(* IEC 61131-3 sources: programs/VI-54/VI-54_20171205/VI-54_20171205/Stations/Screen/LseClass170718/Class/DiagnosticStation, 1 file *)

(* ---- DiagnosticStation.st ---- *)
(*!
<Class
	Name               = "DiagnosticStation"
	Revision           = "1.1"
	RealtimeTask       = "false"
	CyclicTask         = "false"
	BackgroundTask     = "false"
	Sigmatek           = "false"
	OSInterface        = "false"
	HighPriority       = "false"
	Automatic          = "false"
	UpdateMode         = "Prescan"
	SharedCommandTable = "true"
	Objectsize         = "(960,420)"
	Comment            = "Use this class for new stations for the diagnostic export.">
	<Channels>
		<Server Name="ClassSvr" Visualized="false" Initialize="false" WriteProtected="true" Retentive="false" Comment="Is not used."/>
		<Server Name="ID_Destination" Visualized="false" Initialize="true" WriteProtected="true" Retentive="false"/>
		<Server Name="ID_Source" Visualized="false" Initialize="true" WriteProtected="true" Retentive="false"/>
		<Server Name="sStationName" Class="StringInternal" Visualized="false" Initialize="true" WriteProtected="false" Retentive="false" Comment="Name of the station."/>
		<Server Name="sStatus" Visualized="false" Initialize="false" WriteProtected="true" Retentive="false" Comment="Shows the actual state."/>
		<Client Name="cHandler" Required="true" Internal="false" Comment="Object channel to DiagnosticStationHandler."/>
		<Client Name="cPrio" Required="true" Internal="false" Comment="Communication priority number."/>
		<Client Name="cUserFunction" Required="true" Internal="false" Comment="Object channel to UserFunction."/>
		<Client Name="DiagnosticWork" Required="true" Internal="true"/>
		<Client Name="ReceiveDataCMD" Required="true" Internal="true"/>
		<Client Name="SendDataCMD" Required="true" Internal="true"/>
		<Client Name="toDataManager" Required="true" Internal="false" Comment="Connection to communication data manager."/>
	</Channels>
	<RevDoku>
		<Owner Company="Sigmatek"/>
		<Dokumentation Revision="1.1" Date="2016-06-15" Author="HasHan" Company="Sigmatek" Description="changed some clients to server"/>
		<Dokumentation Revision="1.0" Date="2016-06-02" Author="HötAnt" Company="Sigmatek" Description="Creation"/>
	</RevDoku>
	<Network Name="DiagnosticStation">
		<!-- List of Components in this network -->
		<Components>
			<Object
				Name           = "DiagnosticWork"
				Class          = "DiagnosticWork"
				Position       = "(420,120)"
				Visualized     = "false"
				BackgroundTime = "2 ms">
				<Channels>
					<Server Name="sStationName" Value="&quot;PLC1&quot;"/>
					<Server Name="sStatus"/>
					<Client Name="cHandler"/>
					<Client Name="cToCom"/>
					<Client Name="cUserFunction"/>
				</Channels>
			</Object>
			<Object
				Name       = "ReceiveDataCMD"
				Class      = "ReceiveDataCMD"
				Position   = "(360,900)"
				Visualized = "false">
				<Channels>
					<Server Name="ClassSvr"/>
					<Server Name="ID_Source"/>
					<Server Name="sRecvCnt"/>
					<Client Name="cDiagnosticWork"/>
					<Client Name="toDataManager"/>
				</Channels>
			</Object>
			<Object
				Name       = "SendDataCMD"
				Class      = "SendDataCMD"
				Position   = "(390,450)"
				Visualized = "false">
				<Channels>
					<Server Name="ClassSvr"/>
					<Server Name="ID_Destination"/>
					<Server Name="ID_Source"/>
					<Server Name="sSendCnt"/>
					<Server Name="sSendErr"/>
					<Client Name="cPrio"/>
					<Client Name="cStation"/>
					<Client Name="toDataManager"/>
				</Channels>
			</Object>
		</Components>
		<Comments>
		</Comments>
		<!-- List of Connections in this network -->
		<Connections>
			<Connection Source="this.DiagnosticWork" Destination="DiagnosticWork.sStatus"/>
			<Connection Source="this.ID_Destination" Destination="SendDataCMD.ID_Destination" Vertices="(1066,450),(876,600),"/>
			<Connection Source="this.ID_Source" Destination="SendDataCMD.ID_Source" Vertices="(1066,390),(876,660),"/>
			<Connection Source="DiagnosticWork.cHandler" Destination="this.cHandler" Vertices="(420,210),(38,210),"/>
			<Connection Source="DiagnosticWork.cToCom" Destination="SendDataCMD.ClassSvr" Vertices="(420,270),(300,270),(300,390),(930,390),(930,540),(876,540),"/>
			<Connection Source="DiagnosticWork.cUserFunction" Destination="this.cUserFunction" Vertices="(420,330),(38,330),"/>
			<Connection Source="SendDataCMD.cStation" Destination="DiagnosticWork.sStatus" Vertices="(390,660),(870,210),"/>
			<Connection Source="SendDataCMD.cPrio" Destination="this.cPrio" Vertices="(390,600),(38,390),"/>
			<Connection Source="this.sStatus" Destination="DiagnosticWork.sStatus" Vertices="(1066,270),(870,210),"/>
			<Connection Source="this.sStationName" Destination="DiagnosticWork.sStationName" Vertices="(1066,330),(870,270),"/>
			<Connection Source="this.SendDataCMD" Destination="SendDataCMD.ClassSvr"/>
			<Connection Source="SendDataCMD.toDataManager" Destination="this.toDataManager" Vertices="(390,540),(38,270),"/>
			<Connection Source="this.ReceiveDataCMD" Destination="ReceiveDataCMD.ClassSvr"/>
			<Connection Source="ReceiveDataCMD.toDataManager" Destination="this.toDataManager" Vertices="(360,990),(38,270),"/>
			<Connection Source="ReceiveDataCMD.cDiagnosticWork" Destination="DiagnosticWork.sStatus" Vertices="(360,1050),(870,210),"/>
		</Connections>
		<!-- Headerfiles -->
		<Options>
		</Options>
	</Network>
</Class>
*)
DiagnosticStation : CLASS
  //Servers:
	ClassSvr 	: SvrChCmd_DINT;
	sStatus 	: SvrCh_iprStates;
	sStationName 	: SvrChCmd_UDINT;
	ID_Source 	: SvrCh_DINT;
	ID_Destination 	: SvrCh_DINT;
  //Clients:
	DiagnosticWork 	: CltChCmd_DiagnosticWork;
	cHandler 	: CltChCmd_DiagnosticStationHandlerBase;
	toDataManager 	: CltChCmd_DataManager;
	cUserFunction 	: CltChCmd_DiagnosticUserFunction;
	cPrio 	: CltCh_DINT;
	ReceiveDataCMD 	: CltChCmd_ReceiveDataCMD;
	SendDataCMD 	: CltChCmd_SendDataCMD;
  //Variables:
  //Functions:

	FUNCTION VIRTUAL GLOBAL Init;

	FUNCTION VIRTUAL GLOBAL sStatus::Read
		VAR_OUTPUT
			output (EAX) 	: iprStates;
		END_VAR;

	FUNCTION VIRTUAL GLOBAL ID_Source::Read
		VAR_OUTPUT
			output (EAX) 	: DINT;
		END_VAR;

	FUNCTION VIRTUAL GLOBAL ID_Destination::Read
		VAR_OUTPUT
			output (EAX) 	: DINT;
		END_VAR;
  //Tables:
	FUNCTION @STD
		VAR_OUTPUT
			ret_code	: CONFSTATES;
		END_VAR;
	FUNCTION GLOBAL TAB @CT_;
END_CLASS;

#pragma using DiagnosticWork
#pragma using ReceiveDataCMD
#pragma using SendDataCMD
#pragma usingLtd DataManager
#pragma usingLtd DiagnosticStationHandlerBase
#pragma usingLtd DiagnosticUserFunction

FUNCTION VIRTUAL GLOBAL DiagnosticStation::Init

  if _FirstScan then
    ReceiveDataCMD.ID_Source := ID_Source; //set the same ID to the receive-object
  end_if;

END_FUNCTION

FUNCTION VIRTUAL GLOBAL DiagnosticStation::sStatus::Read
	VAR_OUTPUT
		output (EAX) 	: iprStates;
	END_VAR

	sStatus := DiagnosticWork.sStatus.Read();
	output := sStatus;

END_FUNCTION

FUNCTION VIRTUAL GLOBAL DiagnosticStation::ID_Destination::Read
	VAR_OUTPUT
		output (EAX) 	: DINT;
	END_VAR

	ID_Destination := SendDataCMD.ID_Destination.Read();
	output := ID_Destination;

END_FUNCTION

FUNCTION VIRTUAL GLOBAL DiagnosticStation::ID_Source::Read
	VAR_OUTPUT
		output (EAX) 	: DINT;
	END_VAR

	ID_Source := SendDataCMD.ID_Source.Read();
	output := ID_Source;

END_FUNCTION
